// TIA Portal V19 export
FUNCTION "RO PROCESS." : Void   // FC15, LAD
{ S7_Optimized_Access := 'TRUE' }
// stored: SetENOAutomatically false
BEGIN

REGION Network 1: AUTO FLUSHING AV3
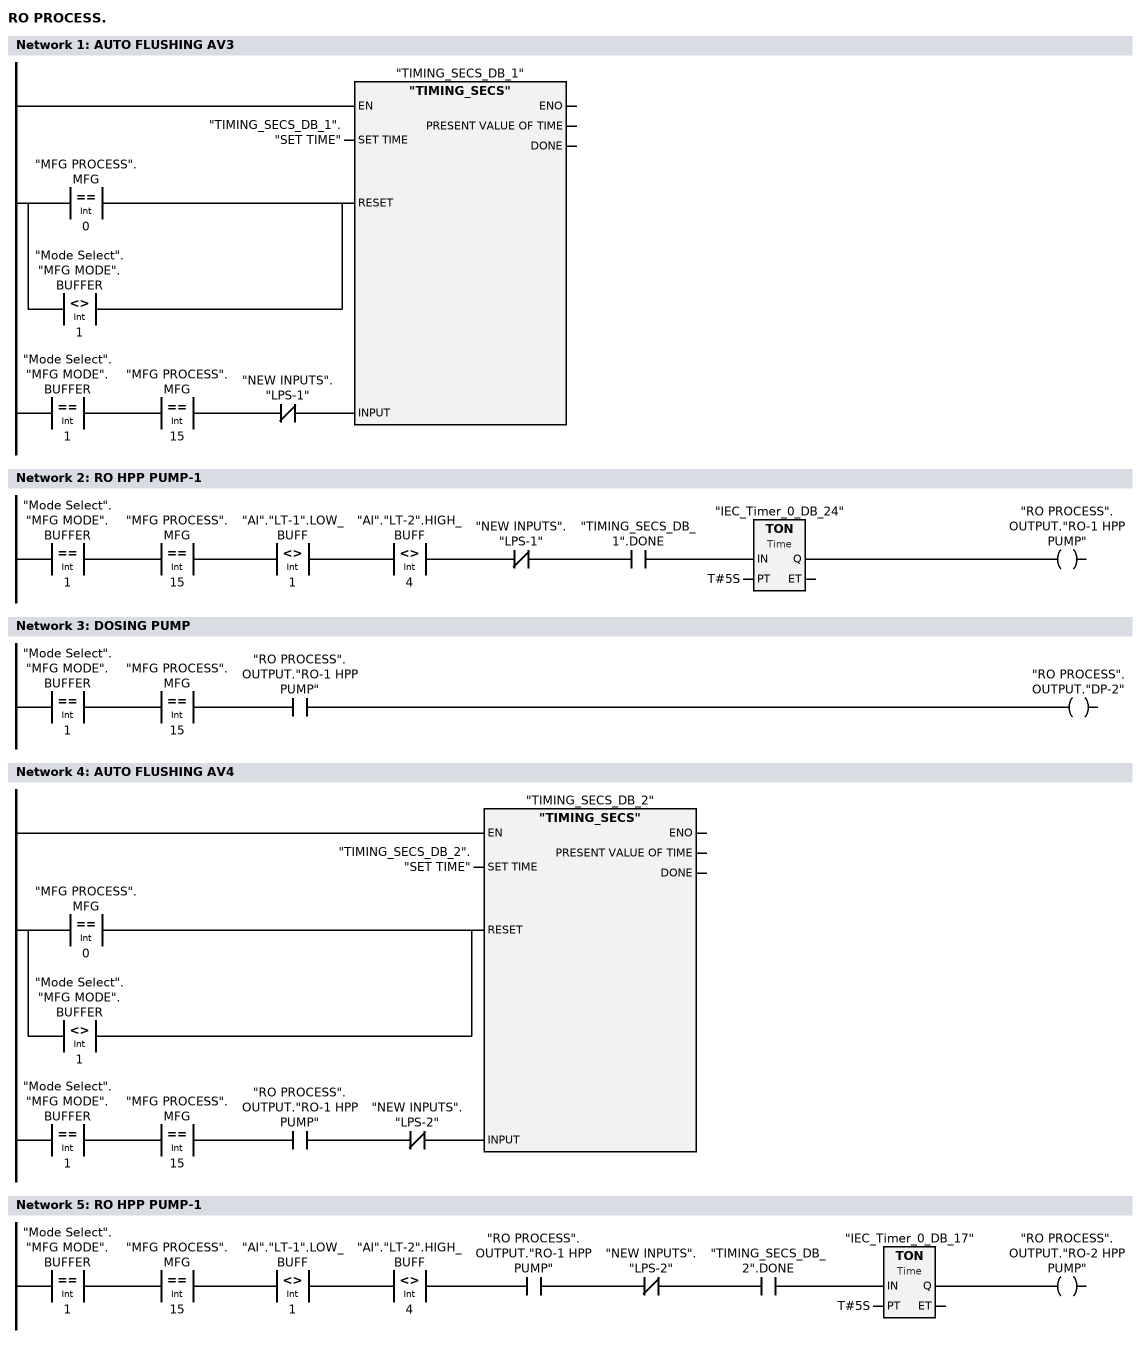
   RUNG wire#powerrail
      "TIMING_SECS_DB_1"(RESET := wire#w1, INPUT := wire#w2, "SET TIME" := "TIMING_SECS_DB_1"."SET TIME", "PRESENT VALUE OF TIME" =>, DONE =>)
   END_RUNG
   RUNG wire#powerrail
      { S7_Templates := "SrcType := Int" } EQ_Contact(in1 := "MFG PROCESS".MFG, in2 := 0)
   END_RUNG wire#w1
   RUNG wire#powerrail
      { S7_Templates := "SrcType := Int" } NE_Contact(in1 := "Mode Select"."MFG MODE".BUFFER, in2 := 1)
   END_RUNG wire#w1
   RUNG wire#powerrail
      { S7_Templates := "SrcType := Int" } EQ_Contact(in1 := "Mode Select"."MFG MODE".BUFFER, in2 := 1)
      { S7_Templates := "SrcType := Int" } EQ_Contact(in1 := "MFG PROCESS".MFG, in2 := 15)
      I_Contact( "NEW INPUTS"."LPS-1" )
   END_RUNG wire#w2
   // the same network as SCL:
   "TIMING_SECS_DB_1"("SET TIME" := "TIMING_SECS_DB_1"."SET TIME",   // "TIMING_SECS"
                      RESET := ("MFG PROCESS".MFG = 0) OR ("Mode Select"."MFG MODE".BUFFER <> 1),
                      INPUT := ("Mode Select"."MFG MODE".BUFFER = 1) AND ("MFG PROCESS".MFG = 15) AND NOT "NEW INPUTS"."LPS-1");
END_REGION

REGION Network 2: RO HPP PUMP-1
   RUNG wire#powerrail
      { S7_Templates := "SrcType := Int" } EQ_Contact(in1 := "Mode Select"."MFG MODE".BUFFER, in2 := 1)
      { S7_Templates := "SrcType := Int" } EQ_Contact(in1 := "MFG PROCESS".MFG, in2 := 15)
      { S7_Templates := "SrcType := Int" } NE_Contact(in1 := "AI"."LT-1".LOW_BUFF, in2 := 1)
      { S7_Templates := "SrcType := Int" } NE_Contact(in1 := "AI"."LT-2".HIGH_BUFF, in2 := 4)
      I_Contact( "NEW INPUTS"."LPS-1" )
      Contact( "TIMING_SECS_DB_1".DONE )
      { S7_Templates := "time_type := Time" } "IEC_Timer_0_DB_24".TON(pt := T#5S, et =>)
      Coil( "RO PROCESS".OUTPUT."RO-1 HPP PUMP" )
   END_RUNG
   // the same network as SCL:
   "IEC_Timer_0_DB_24".TON(IN := ("Mode Select"."MFG MODE".BUFFER = 1) AND ("MFG PROCESS".MFG = 15) AND ("AI"."LT-1".LOW_BUFF <> 1) AND ("AI"."LT-2".HIGH_BUFF <> 4) AND NOT "NEW INPUTS"."LPS-1" AND "TIMING_SECS_DB_1".DONE,
                           PT := T#5S);
   "RO PROCESS".OUTPUT."RO-1 HPP PUMP" := "IEC_Timer_0_DB_24".Q;
END_REGION

REGION Network 3: DOSING PUMP
   RUNG wire#powerrail
      { S7_Templates := "SrcType := Int" } EQ_Contact(in1 := "Mode Select"."MFG MODE".BUFFER, in2 := 1)
      { S7_Templates := "SrcType := Int" } EQ_Contact(in1 := "MFG PROCESS".MFG, in2 := 15)
      Contact( "RO PROCESS".OUTPUT."RO-1 HPP PUMP" )
      Coil( "RO PROCESS".OUTPUT."DP-2" )
   END_RUNG
   // the same network as SCL:
   "RO PROCESS".OUTPUT."DP-2" := ("Mode Select"."MFG MODE".BUFFER = 1) AND ("MFG PROCESS".MFG = 15) AND "RO PROCESS".OUTPUT."RO-1 HPP PUMP";
END_REGION

REGION Network 4: AUTO FLUSHING AV4
   RUNG wire#powerrail
      "TIMING_SECS_DB_2"(RESET := wire#w1, INPUT := wire#w2, "SET TIME" := "TIMING_SECS_DB_2"."SET TIME", "PRESENT VALUE OF TIME" =>, DONE =>)
   END_RUNG
   RUNG wire#powerrail
      { S7_Templates := "SrcType := Int" } EQ_Contact(in1 := "MFG PROCESS".MFG, in2 := 0)
   END_RUNG wire#w1
   RUNG wire#powerrail
      { S7_Templates := "SrcType := Int" } NE_Contact(in1 := "Mode Select"."MFG MODE".BUFFER, in2 := 1)
   END_RUNG wire#w1
   RUNG wire#powerrail
      { S7_Templates := "SrcType := Int" } EQ_Contact(in1 := "Mode Select"."MFG MODE".BUFFER, in2 := 1)
      { S7_Templates := "SrcType := Int" } EQ_Contact(in1 := "MFG PROCESS".MFG, in2 := 15)
      Contact( "RO PROCESS".OUTPUT."RO-1 HPP PUMP" )
      I_Contact( "NEW INPUTS"."LPS-2" )
   END_RUNG wire#w2
   // the same network as SCL:
   "TIMING_SECS_DB_2"("SET TIME" := "TIMING_SECS_DB_2"."SET TIME",   // "TIMING_SECS"
                      RESET := ("MFG PROCESS".MFG = 0) OR ("Mode Select"."MFG MODE".BUFFER <> 1),
                      INPUT := ("Mode Select"."MFG MODE".BUFFER = 1) AND ("MFG PROCESS".MFG = 15) AND "RO PROCESS".OUTPUT."RO-1 HPP PUMP" AND NOT "NEW INPUTS"."LPS-2");
END_REGION

REGION Network 5: RO HPP PUMP-1
   RUNG wire#powerrail
      { S7_Templates := "SrcType := Int" } EQ_Contact(in1 := "Mode Select"."MFG MODE".BUFFER, in2 := 1)
      { S7_Templates := "SrcType := Int" } EQ_Contact(in1 := "MFG PROCESS".MFG, in2 := 15)
      { S7_Templates := "SrcType := Int" } NE_Contact(in1 := "AI"."LT-1".LOW_BUFF, in2 := 1)
      { S7_Templates := "SrcType := Int" } NE_Contact(in1 := "AI"."LT-2".HIGH_BUFF, in2 := 4)
      Contact( "RO PROCESS".OUTPUT."RO-1 HPP PUMP" )
      I_Contact( "NEW INPUTS"."LPS-2" )
      Contact( "TIMING_SECS_DB_2".DONE )
      { S7_Templates := "time_type := Time" } "IEC_Timer_0_DB_17".TON(pt := T#5S, et =>)
      Coil( "RO PROCESS".OUTPUT."RO-2 HPP PUMP" )
   END_RUNG
   // the same network as SCL:
   "IEC_Timer_0_DB_17".TON(IN := ("Mode Select"."MFG MODE".BUFFER = 1) AND ("MFG PROCESS".MFG = 15) AND ("AI"."LT-1".LOW_BUFF <> 1) AND ("AI"."LT-2".HIGH_BUFF <> 4) AND "RO PROCESS".OUTPUT."RO-1 HPP PUMP" AND NOT "NEW INPUTS"."LPS-2" AND "TIMING_SECS_DB_2".DONE,
                           PT := T#5S);
   "RO PROCESS".OUTPUT."RO-2 HPP PUMP" := "IEC_Timer_0_DB_17".Q;
END_REGION
END_FUNCTION
